// TwinCAT 3 PLC project Sample01
// ProgramVersion: 3.1.4022.7
// libraries:
//   Tc2_Standard, * (Beckhoff Automation GmbH)
//   Tc2_System, * (Beckhoff Automation GmbH)
//   Tc3_Module, * (Beckhoff Automation GmbH)
// project tree:
//   / PlcTask.TcTTO
//   POUs/ F_Calc.TcPOU, MAIN.TcPOU
// real-time tasks:
//   TASK PlcTask: cycle T#10ms, priority 20, ADS port 350

CONFIGURATION Sample01
    RESOURCE PLC ON TwinCAT3
        TASK PlcTask(INTERVAL := T#10ms, PRIORITY := 20);
        PROGRAM MAIN WITH PlcTask : MAIN;
    END_RESOURCE
END_CONFIGURATION

// ---- POUs/MAIN.TcPOU
PROGRAM MAIN
VAR
	aData		: ARRAY[0..9] OF LREAL := [0, 1, 2, 3, 4, 5, 6, 7, 8, 9];
	fValue		: LREAL;
END_VAR

fValue := F_Calc(ADR(aData), 1, 2);

END_PROGRAM

// ---- POUs/F_Calc.TcPOU
FUNCTION F_Calc : LREAL
VAR_INPUT
	pData		: POINTER TO ARRAY [0..9] OF LREAL;
	nElementA	: INT;
	nElementB 	: INT;
END_VAR
VAR
	exc			: __SYSTEM.ExceptionCode;
END_VAR

__TRY
	F_Calc := pData^[nElementA] / pData^[nElementB];
__CATCH (exc)
	IF (exc = __SYSTEM.ExceptionCode.RTSEXCPT_ARRAYBOUNDS) THEN
		F_Calc := -1;
    ELSIF ((exc = __SYSTEM.ExceptionCode.RTSEXCPT_FPU_DIVIDEBYZERO) OR
	       (exc = __SYSTEM.ExceptionCode.RTSEXCPT_DIVIDEBYZERO)) THEN
		F_Calc := -2;
	ELSIF (exc = __SYSTEM.ExceptionCode.RTSEXCPT_ACCESS_VIOLATION) THEN
		F_Calc := -3;
	ELSE
		F_Calc := -4;
	END_IF
__FINALLY
	F_Calc := F_Calc + 1;
__ENDTRY

END_FUNCTION
